// Mitsubishi GX Works2 project: 大成外環大泉FLEX   PLC: Q02/Q02H

PROGRAM FLEXPIWI  // PID演算 for WIndows
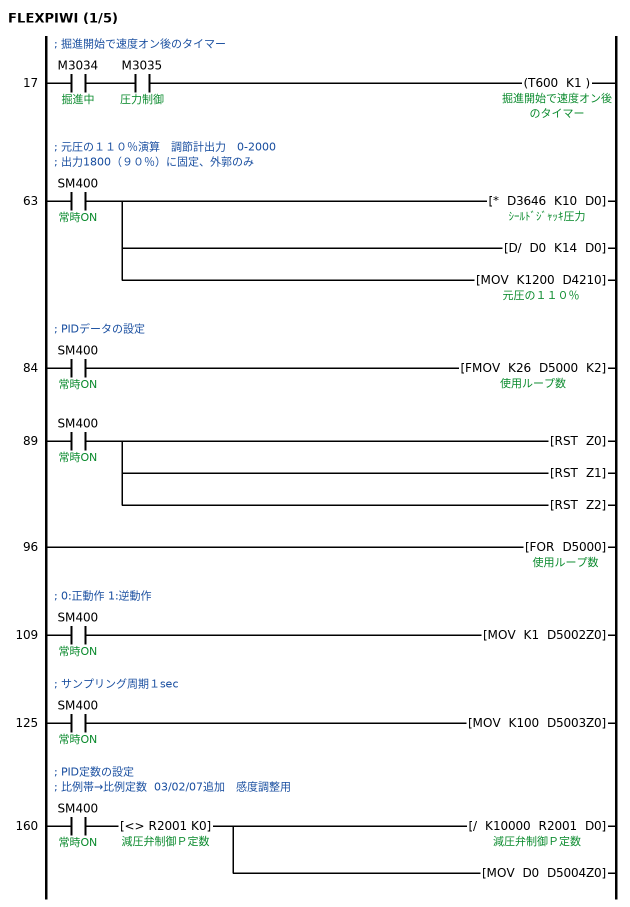
; 掘進開始で速度オン後のタイマー
17    LD      M3034  ; 掘進中
      AND     M3035  ; 圧力制御
      OUT     T600 K1  ; 掘進開始で速度オン後のタイマー
; 元圧の１１０％演算　調節計出力　0-2000
; 出力1800（９０％）に固定、外郭のみ
63    LD      SM400  ; 常時ON
      *       D3646 K10 D0  ; ｼｰﾙﾄﾞｼﾞｬｯｷ圧力
      D/      D0 K14 D0
      MOV     K1200 D4210  ; 元圧の１１０％
; PIDデータの設定
84    LD      SM400  ; 常時ON
      FMOV    K26 D5000 K2  ; 使用ループ数
89    LD      SM400  ; 常時ON
      RST     Z0
      RST     Z1
      RST     Z2
96    FOR     D5000
; 0:正動作 1:逆動作
109   LD      SM400  ; 常時ON
      MOV     K1 D5002Z0
; サンプリング周期１sec
125   LD      SM400  ; 常時ON
      MOV     K100 D5003Z0
; PID定数の設定
; 比例帯→比例定数  03/02/07追加　感度調整用
160   LD      SM400  ; 常時ON
      AND<>   R2001 K0  ; 減圧弁制御Ｐ定数
      /       K10000 R2001 D0
      MOV     D0 D5004Z0
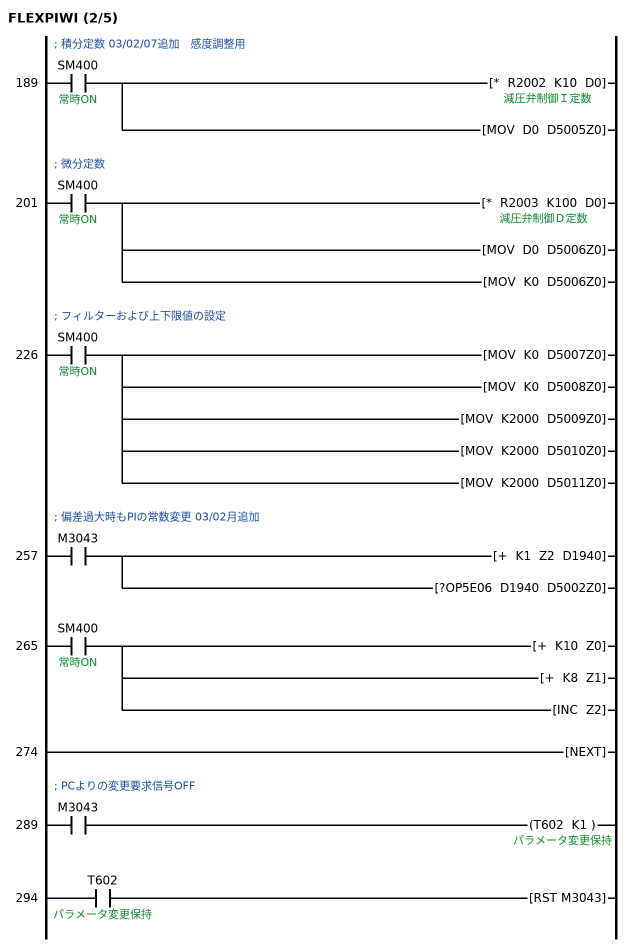
; 積分定数 03/02/07追加　感度調整用
189   LD      SM400  ; 常時ON
      *       R2002 K10 D0  ; 減圧弁制御Ｉ定数
      MOV     D0 D5005Z0
; 微分定数
201   LD      SM400  ; 常時ON
      *       R2003 K100 D0  ; 減圧弁制御Ｄ定数
      MOV     D0 D5006Z0
      MOV     K0 D5006Z0
; フィルターおよび上下限値の設定
226   LD      SM400  ; 常時ON
      MOV     K0 D5007Z0
      MOV     K0 D5008Z0
      MOV     K2000 D5009Z0
      MOV     K2000 D5010Z0
      MOV     K2000 D5011Z0
; 偏差過大時もPIの常数変更 03/02月追加
257   LD      M3043
      +       K1 Z2 D1940
      ?OP5E06 D1940 D5002Z0
265   LD      SM400  ; 常時ON
      +       K10 Z0
      +       K8 Z1
      INC     Z2
274   NEXT
; PCよりの変更要求信号OFF
289   LD      M3043
      OUT     T602 K1  ; パラメータ変更保持
294   LD      T602  ; パラメータ変更保持
      RST     M3043
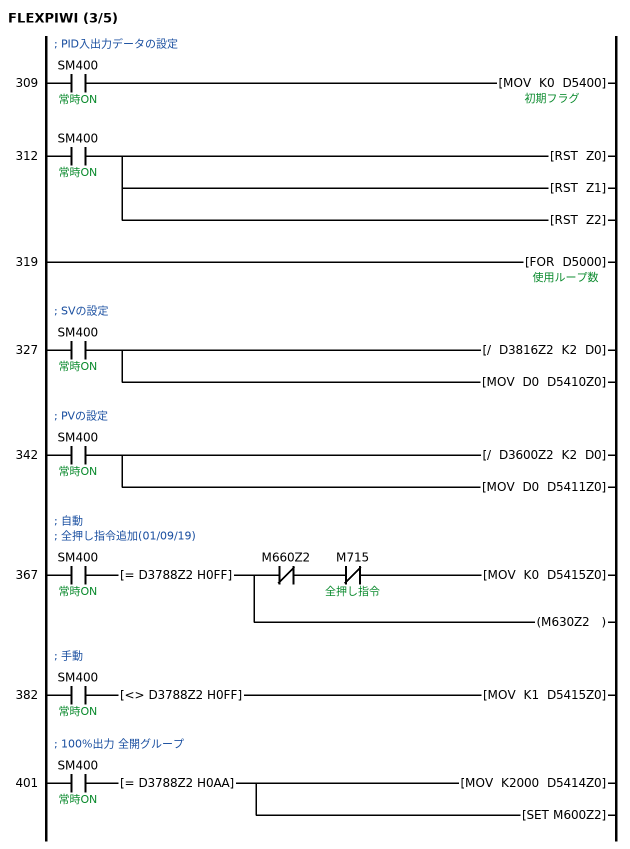
; PID入出力データの設定
309   LD      SM400  ; 常時ON
      MOV     K0 D5400  ; 初期フラグ
312   LD      SM400  ; 常時ON
      RST     Z0
      RST     Z1
      RST     Z2
319   FOR     D5000
; SVの設定
327   LD      SM400  ; 常時ON
      /       D3816Z2 K2 D0
      MOV     D0 D5410Z0
; 
; PVの設定
342   LD      SM400  ; 常時ON
      /       D3600Z2 K2 D0
      MOV     D0 D5411Z0
; 自動
; 全押し指令追加(01/09/19)
367   LD      SM400  ; 常時ON
      AND=    D3788Z2 H0FF
      MPS
      ANI     M660Z2
      ANI     M715  ; 全押し指令
      MOV     K0 D5415Z0
      MPP
      OUT     M630Z2
; 手動
382   LD      SM400  ; 常時ON
      AND<>   D3788Z2 H0FF
      MOV     K1 D5415Z0
; 100%出力 全開グループ
401   LD      SM400  ; 常時ON
      AND=    D3788Z2 H0AA
      MOV     K2000 D5414Z0
      SET     M600Z2
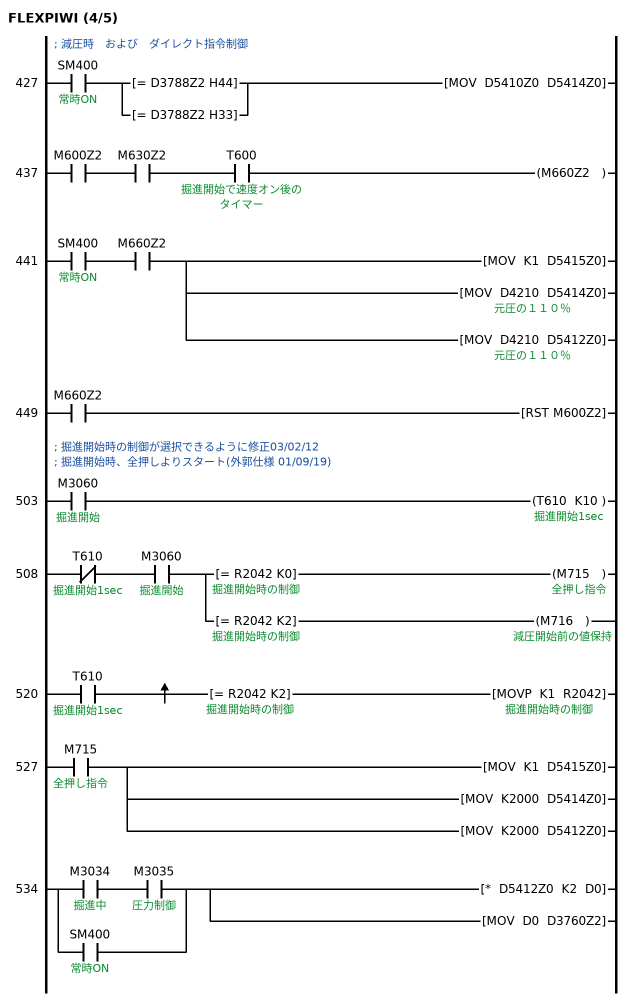
; 減圧時　および　ダイレクト指令制御
427   LD      SM400  ; 常時ON
      LD=     D3788Z2 H44
      OR=     D3788Z2 H33
      ANB
      MOV     D5410Z0 D5414Z0
437   LD      M600Z2
      AND     M630Z2
      AND     T600  ; 掘進開始で速度オン後のタイマー
      OUT     M660Z2
441   LD      SM400  ; 常時ON
      AND     M660Z2
      MOV     K1 D5415Z0
      MOV     D4210 D5414Z0
      MOV     D4210 D5412Z0
449   LD      M660Z2
      RST     M600Z2
; 掘進開始時の制御が選択できるように修正03/02/12
; 掘進開始時、全押しよりスタート(外郭仕様 01/09/19)
503   LD      M3060  ; 掘進開始
      OUT     T610 K10  ; 掘進開始1sec
508   LDI     T610  ; 掘進開始1sec
      AND     M3060  ; 掘進開始
      MPS
      AND=    R2042 K0  ; 掘進開始時の制御
      OUT     M715  ; 全押し指令
      MPP
      AND=    R2042 K2  ; 掘進開始時の制御
      OUT     M716  ; 減圧開始前の値保持
520   LD      T610  ; 掘進開始1sec
      MEP
      AND=    R2042 K2  ; 掘進開始時の制御
      MOVP    K1 R2042
527   LD      M715  ; 全押し指令
      MOV     K1 D5415Z0
      MOV     K2000 D5414Z0
      MOV     K2000 D5412Z0
534   LD      M3034  ; 掘進中
      AND     M3035  ; 圧力制御
      OR      SM400  ; 常時ON
      *       D5412Z0 K2 D0
      MOV     D0 D3760Z2
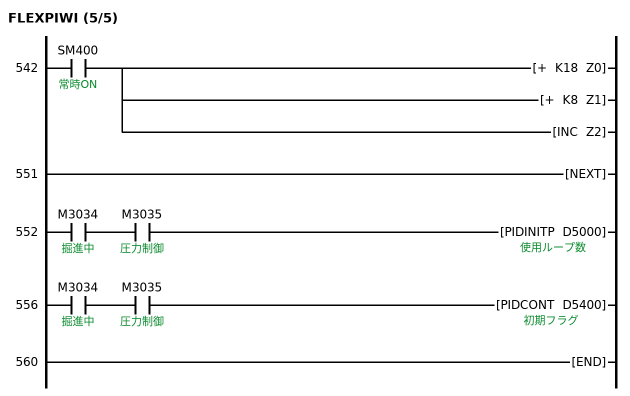
542   LD      SM400  ; 常時ON
      +       K18 Z0
      +       K8 Z1
      INC     Z2
551   NEXT
552   LD      M3034  ; 掘進中
      AND     M3035  ; 圧力制御
      PIDINITP D5000
556   LD      M3034  ; 掘進中
      AND     M3035  ; 圧力制御
      PIDCONT D5400
560   END
END_PROGRAM

PROGRAM FLEXWIN  // FlexWindos対応
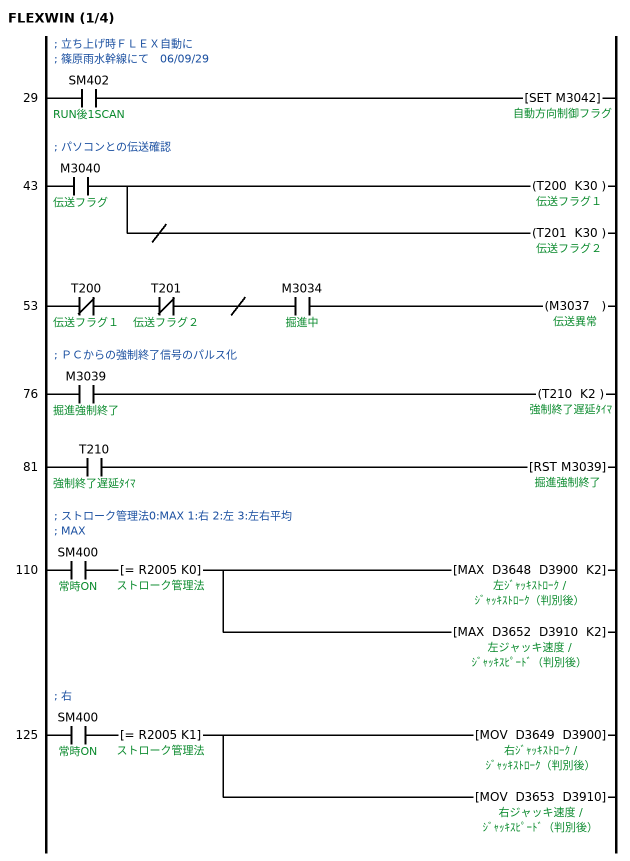
; 立ち上げ時ＦＬＥＸ自動に
; 篠原雨水幹線にて　06/09/29
29    LD      SM402  ; RUN後1SCAN
      SET     M3042  ; 自動方向制御フラグ
; パソコンとの伝送確認
43    LD      M3040  ; 伝送フラグ
      OUT     T200 K30  ; 伝送フラグ１
      INV
      OUT     T201 K30  ; 伝送フラグ２
53    LDI     T200  ; 伝送フラグ１
      ANI     T201  ; 伝送フラグ２
      INV
      AND     M3034  ; 掘進中
      OUT     M3037  ; 伝送異常
; ＰＣからの強制終了信号のパルス化
76    LD      M3039  ; 掘進強制終了
      OUT     T210 K2  ; 強制終了遅延ﾀｲﾏ
81    LD      T210  ; 強制終了遅延ﾀｲﾏ
      RST     M3039  ; 掘進強制終了
; ストローク管理法0:MAX 1:右 2:左 3:左右平均
; MAX
110   LD      SM400  ; 常時ON
      AND=    R2005 K0  ; ストローク管理法
      MAX     D3648 D3900 K2  ; 左ｼﾞｬｯｷｽﾄﾛｰｸ / ｼﾞｬｯｷｽﾄﾛｰｸ（判別後）
      MAX     D3652 D3910 K2  ; 左ジャッキ速度 / ｼﾞｬｯｷｽﾋﾟｰﾄﾞ（判別後）
; 右
125   LD      SM400  ; 常時ON
      AND=    R2005 K1  ; ストローク管理法
      MOV     D3649 D3900  ; 右ｼﾞｬｯｷｽﾄﾛｰｸ
      MOV     D3653 D3910  ; 右ジャッキ速度
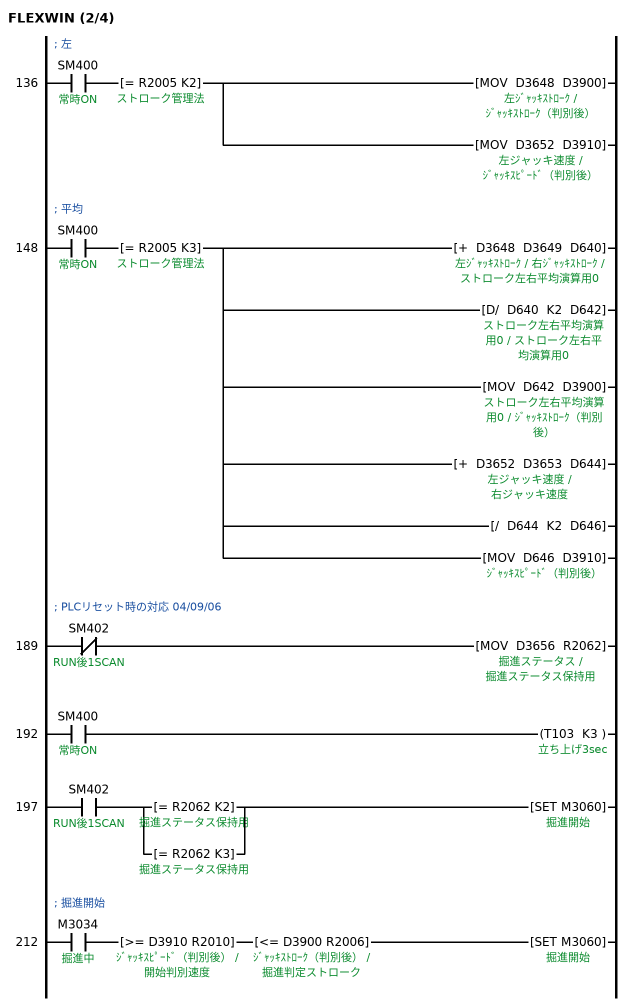
; 左
136   LD      SM400  ; 常時ON
      AND=    R2005 K2  ; ストローク管理法
      MOV     D3648 D3900
      MOV     D3652 D3910
; 平均
148   LD      SM400  ; 常時ON
      AND=    R2005 K3  ; ストローク管理法
      +       D3648 D3649 D640  ; ストローク左右平均演算用0
      D/      D640 K2 D642  ; ストローク左右平均演算用0
      MOV     D642 D3900
      +       D3652 D3653 D644
      /       D644 K2 D646
      MOV     D646 D3910
; PLCリセット時の対応 04/09/06
189   LDI     SM402  ; RUN後1SCAN
      MOV     D3656 R2062  ; 掘進ステータス / 掘進ステータス保持用
192   LD      SM400  ; 常時ON
      OUT     T103 K3  ; 立ち上げ3sec
197   LD      SM402  ; RUN後1SCAN
      LD=     R2062 K2  ; 掘進ステータス保持用
      OR=     R2062 K3  ; 掘進ステータス保持用
      ANB
      SET     M3060  ; 掘進開始
; 掘進開始
212   LD      M3034  ; 掘進中
      AND>=   D3910 R2010  ; ｼﾞｬｯｷｽﾋﾟｰﾄﾞ（判別後） / 開始判別速度
      AND<=   D3900 R2006  ; ｼﾞｬｯｷｽﾄﾛｰｸ（判別後） / 掘進判定ストローク
      SET     M3060  ; 掘進開始
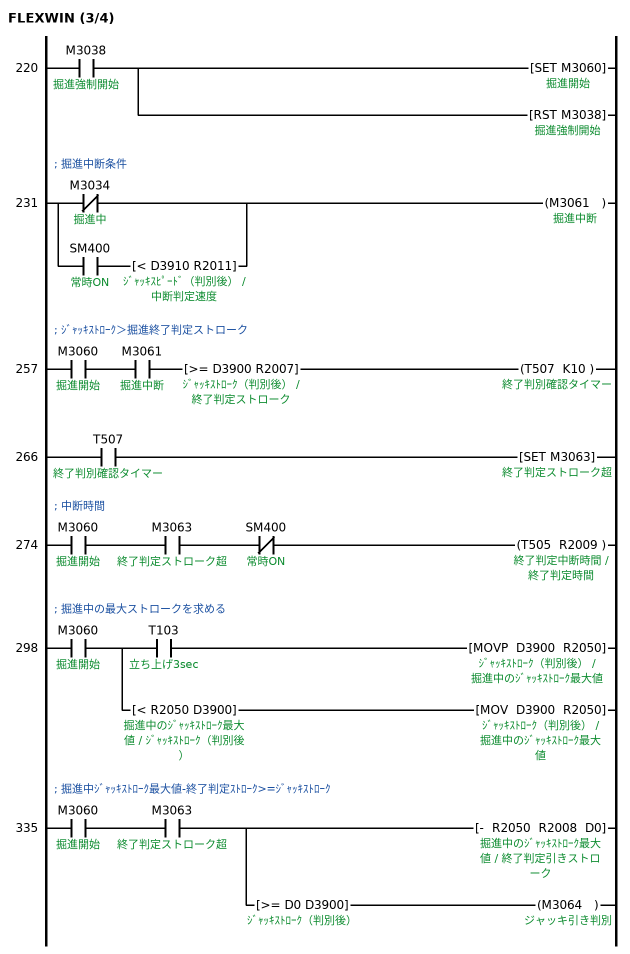
220   LD      M3038  ; 掘進強制開始
      SET     M3060  ; 掘進開始
      RST     M3038  ; 掘進強制開始
; 掘進中断条件
231   LDI     M3034  ; 掘進中
      LD      SM400  ; 常時ON
      AND<    D3910 R2011  ; ｼﾞｬｯｷｽﾋﾟｰﾄﾞ（判別後） / 中断判定速度
      ORB
      OUT     M3061  ; 掘進中断
; ｼﾞｬｯｷｽﾄﾛｰｸ＞掘進終了判定ストローク
257   LD      M3060  ; 掘進開始
      AND     M3061  ; 掘進中断
      AND>=   D3900 R2007  ; ｼﾞｬｯｷｽﾄﾛｰｸ（判別後） / 終了判定ストローク
      OUT     T507 K10  ; 終了判別確認タイマー
266   LD      T507  ; 終了判別確認タイマー
      SET     M3063  ; 終了判定ストローク超
; 中断時間
274   LD      M3060  ; 掘進開始
      AND     M3063  ; 終了判定ストローク超
      ANI     SM400  ; 常時ON
      OUT     T505 R2009  ; 終了判定中断時間 / 終了判定時間
; 掘進中の最大ストロークを求める
298   LD      M3060  ; 掘進開始
      MPS
      AND     T103  ; 立ち上げ3sec
      MOVP    D3900 R2050  ; 掘進中のｼﾞｬｯｷｽﾄﾛｰｸ最大値
      MPP
      AND<    R2050 D3900  ; 掘進中のｼﾞｬｯｷｽﾄﾛｰｸ最大値 / ｼﾞｬｯｷｽﾄﾛｰｸ（判別後）
      MOV     D3900 R2050
; 掘進中ｼﾞｬｯｷｽﾄﾛｰｸ最大値-終了判定ｽﾄﾛｰｸ>=ｼﾞｬｯｷｽﾄﾛｰｸ
335   LD      M3060  ; 掘進開始
      AND     M3063  ; 終了判定ストローク超
      -       R2050 R2008 D0  ; 終了判定引きストローク
      AND>=   D0 D3900  ; ｼﾞｬｯｷｽﾄﾛｰｸ（判別後）
      OUT     M3064  ; ジャッキ引き判別
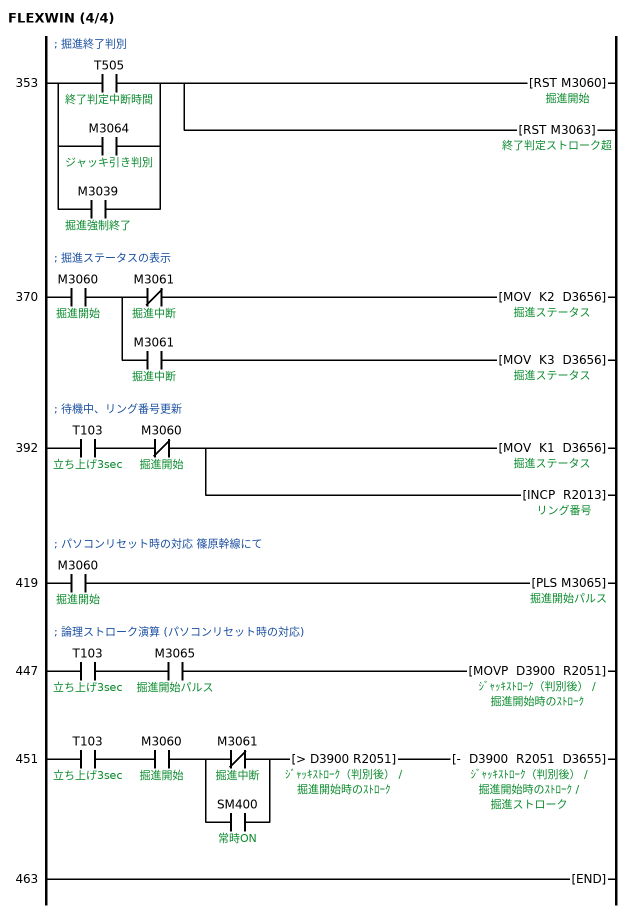
; 掘進終了判別
353   LD      T505  ; 終了判定中断時間
      OR      M3064  ; ジャッキ引き判別
      OR      M3039  ; 掘進強制終了
      RST     M3060  ; 掘進開始
      RST     M3063  ; 終了判定ストローク超
; 掘進ステータスの表示
370   LD      M3060  ; 掘進開始
      MPS
      ANI     M3061  ; 掘進中断
      MOV     K2 D3656
      MPP
      AND     M3061  ; 掘進中断
      MOV     K3 D3656
; 待機中、リング番号更新
392   LD      T103  ; 立ち上げ3sec
      ANI     M3060  ; 掘進開始
      MOV     K1 D3656
      INCP    R2013  ; リング番号
; パソコンリセット時の対応 篠原幹線にて
419   LD      M3060  ; 掘進開始
      PLS     M3065  ; 掘進開始パルス
; 論理ストローク演算 (パソコンリセット時の対応)
447   LD      T103  ; 立ち上げ3sec
      AND     M3065  ; 掘進開始パルス
      MOVP    D3900 R2051  ; 掘進開始時のｽﾄﾛｰｸ
451   LD      T103  ; 立ち上げ3sec
      AND     M3060  ; 掘進開始
      LDI     M3061  ; 掘進中断
      OR      SM400  ; 常時ON
      ANB
      AND>    D3900 R2051  ; ｼﾞｬｯｷｽﾄﾛｰｸ（判別後） / 掘進開始時のｽﾄﾛｰｸ
      -       D3900 R2051 D3655  ; 掘進ストローク
463   END
END_PROGRAM

PROGRAM INOUTWIN  // 大成外環大泉FLEX
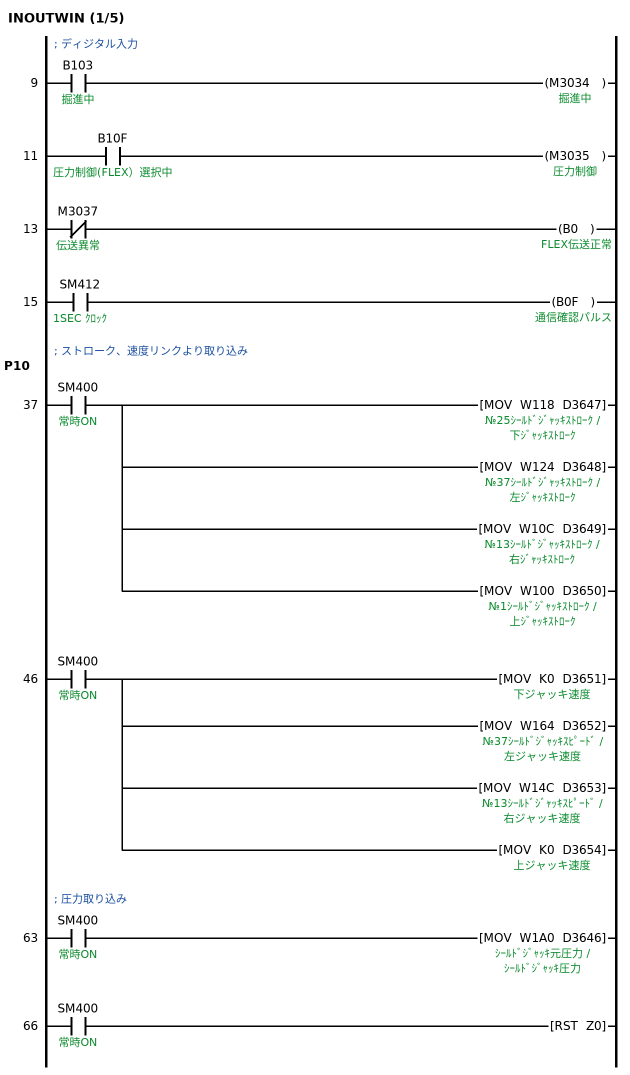
; ディジタル入力
9     LD      B103  ; 掘進中
      OUT     M3034  ; 掘進中
11    LD      B10F  ; 圧力制御(FLEX）選択中
      OUT     M3035  ; 圧力制御
13    LDI     M3037  ; 伝送異常
      OUT     B0  ; FLEX伝送正常
15    LD      SM412  ; 1SEC ｸﾛｯｸ
      OUT     B0F  ; 通信確認パルス
; ストローク、速度リンクより取り込み
      P10
37    LD      SM400  ; 常時ON
      MOV     W118 D3647  ; №25ｼｰﾙﾄﾞｼﾞｬｯｷｽﾄﾛｰｸ / 下ｼﾞｬｯｷｽﾄﾛｰｸ
      MOV     W124 D3648  ; №37ｼｰﾙﾄﾞｼﾞｬｯｷｽﾄﾛｰｸ / 左ｼﾞｬｯｷｽﾄﾛｰｸ
      MOV     W10C D3649  ; №13ｼｰﾙﾄﾞｼﾞｬｯｷｽﾄﾛｰｸ / 右ｼﾞｬｯｷｽﾄﾛｰｸ
      MOV     W100 D3650  ; №1ｼｰﾙﾄﾞｼﾞｬｯｷｽﾄﾛｰｸ / 上ｼﾞｬｯｷｽﾄﾛｰｸ
46    LD      SM400  ; 常時ON
      MOV     K0 D3651  ; 下ジャッキ速度
      MOV     W164 D3652  ; №37ｼｰﾙﾄﾞｼﾞｬｯｷｽﾋﾟｰﾄﾞ / 左ジャッキ速度
      MOV     W14C D3653  ; №13ｼｰﾙﾄﾞｼﾞｬｯｷｽﾋﾟｰﾄﾞ / 右ジャッキ速度
      MOV     K0 D3654  ; 上ジャッキ速度
; 圧力取り込み
63    LD      SM400  ; 常時ON
      MOV     W1A0 D3646  ; ｼｰﾙﾄﾞｼﾞｬｯｷ元圧力 / ｼｰﾙﾄﾞｼﾞｬｯｷ圧力
66    LD      SM400  ; 常時ON
      RST     Z0
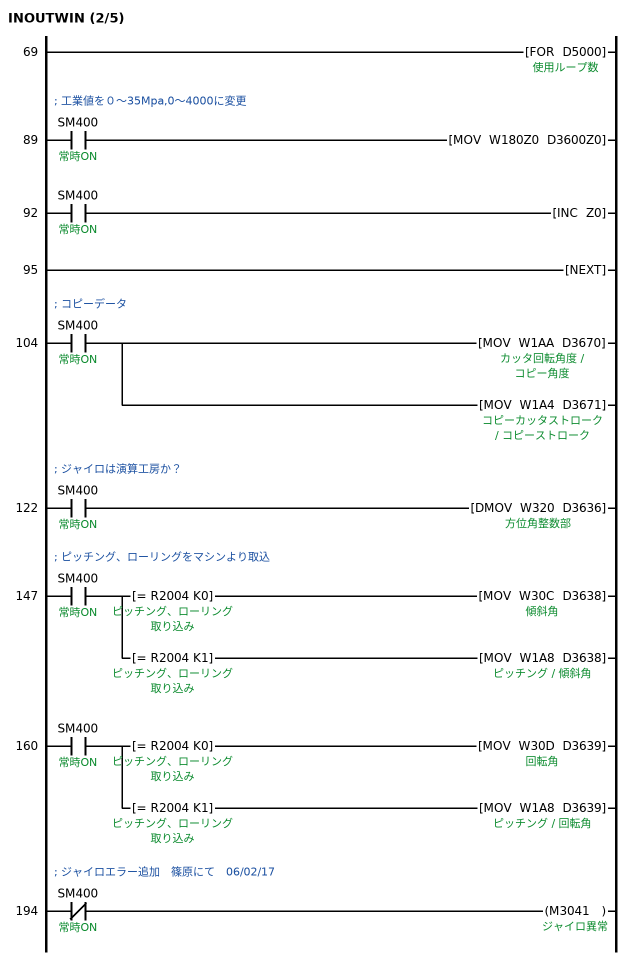
69    FOR     D5000  ; 使用ループ数
; 工業値を０～35Mpa,0～4000に変更
89    LD      SM400  ; 常時ON
      MOV     W180Z0 D3600Z0
92    LD      SM400  ; 常時ON
      INC     Z0
95    NEXT
; コピーデータ
104   LD      SM400  ; 常時ON
      MOV     W1AA D3670  ; カッタ回転角度 / コピー角度
      MOV     W1A4 D3671  ; コピーカッタストローク / コピーストローク
; ジャイロは演算工房か？
122   LD      SM400  ; 常時ON
      DMOV    W320 D3636  ; 方位角整数部
; ピッチング、ローリングをマシンより取込
147   LD      SM400  ; 常時ON
      MPS
      AND=    R2004 K0  ; ピッチング、ローリング取り込み
      MOV     W30C D3638  ; 傾斜角
      MPP
      AND=    R2004 K1  ; ピッチング、ローリング取り込み
      MOV     W1A8 D3638  ; ピッチング
160   LD      SM400  ; 常時ON
      MPS
      AND=    R2004 K0  ; ピッチング、ローリング取り込み
      MOV     W30D D3639  ; 回転角
      MPP
      AND=    R2004 K1  ; ピッチング、ローリング取り込み
      MOV     W1A8 D3639
; ジャイロエラー追加　篠原にて　06/02/17
194   LDI     SM400  ; 常時ON
      OUT     M3041  ; ジャイロ異常
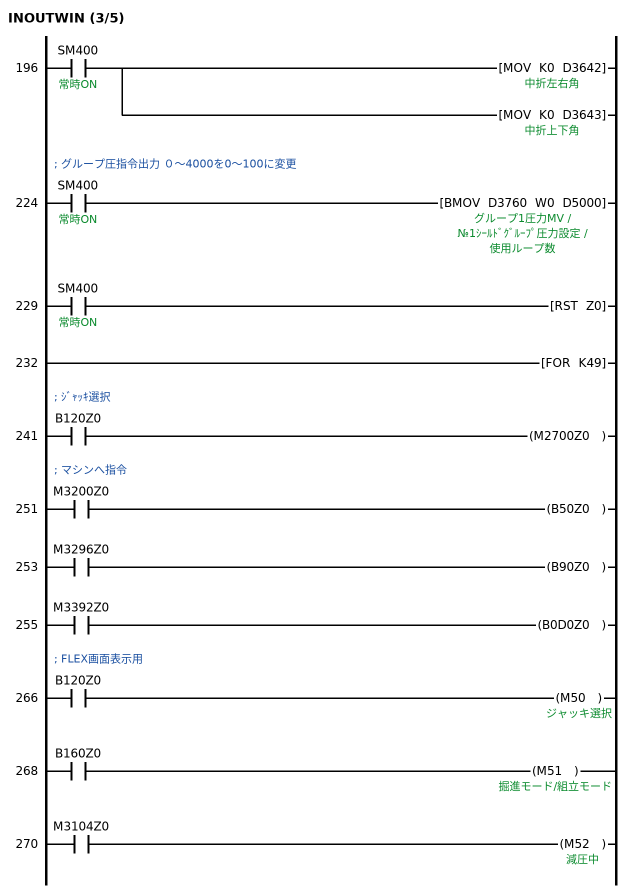
196   LD      SM400  ; 常時ON
      MOV     K0 D3642  ; 中折左右角
      MOV     K0 D3643  ; 中折上下角
; グループ圧指令出力 ０～4000を0～100に変更
224   LD      SM400  ; 常時ON
      BMOV    D3760 W0 D5000  ; グループ1圧力MV / №1ｼｰﾙﾄﾞｸﾞﾙｰﾌﾟ圧力設定
229   LD      SM400  ; 常時ON
      RST     Z0
232   FOR     K49
; ｼﾞｬｯｷ選択
241   LD      B120Z0
      OUT     M2700Z0
; マシンへ指令
251   LD      M3200Z0
      OUT     B50Z0
253   LD      M3296Z0
      OUT     B90Z0
255   LD      M3392Z0
      OUT     B0D0Z0
; FLEX画面表示用
266   LD      B120Z0
      OUT     M50  ; ジャッキ選択
268   LD      B160Z0
      OUT     M51  ; 掘進モード/組立モード
270   LD      M3104Z0
      OUT     M52  ; 減圧中
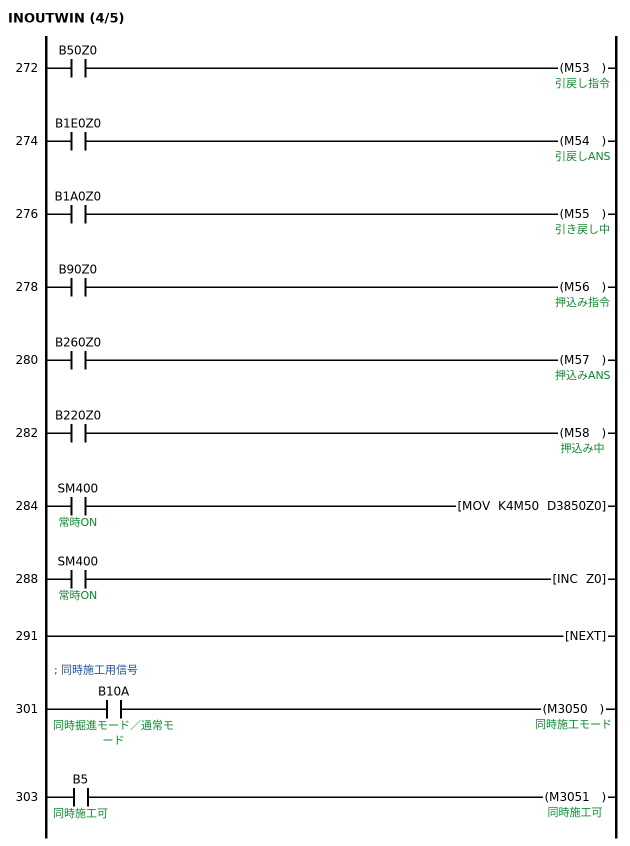
272   LD      B50Z0
      OUT     M53  ; 引戻し指令
274   LD      B1E0Z0
      OUT     M54  ; 引戻しANS
276   LD      B1A0Z0
      OUT     M55  ; 引き戻し中
278   LD      B90Z0
      OUT     M56  ; 押込み指令
280   LD      B260Z0
      OUT     M57  ; 押込みANS
282   LD      B220Z0
      OUT     M58  ; 押込み中
284   LD      SM400  ; 常時ON
      MOV     K4M50 D3850Z0
288   LD      SM400  ; 常時ON
      INC     Z0
291   NEXT
; 同時施工用信号
301   LD      B10A  ; 同時掘進モード／通常モード
      OUT     M3050  ; 同時施工モード
303   LD      B5  ; 同時施工可
      OUT     M3051  ; 同時施工可
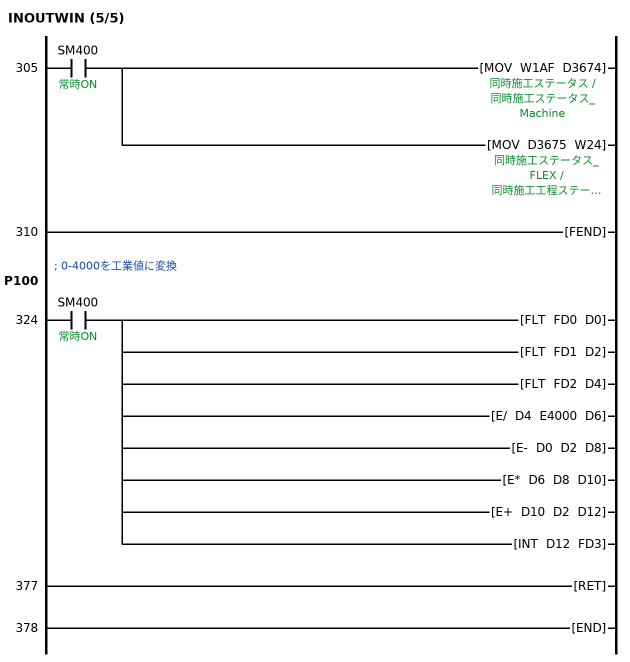
305   LD      SM400  ; 常時ON
      MOV     W1AF D3674  ; 同時施工ステータス / 同時施工ステータス_Machine
      MOV     D3675 W24  ; 同時施工ステータス_FLEX / 同時施工工程ステータス
310   FEND
      P100
; 0-4000を工業値に変換
324   LD      SM400  ; 常時ON
      FLT     FD0 D0
        [note] スケール上限
      FLT     FD1 D2
        [note] スケール下限
      FLT     FD2 D4
        [note] 元アドレス
      E/      D4 E4000 D6
      E-      D0 D2 D8
      E*      D6 D8 D10
      E+      D10 D2 D12
      INT     D12 FD3
377   RET
378   END
END_PROGRAM

PROGRAM TOKIMEC  // ジャイロとの通信 QJ71C24Nタ
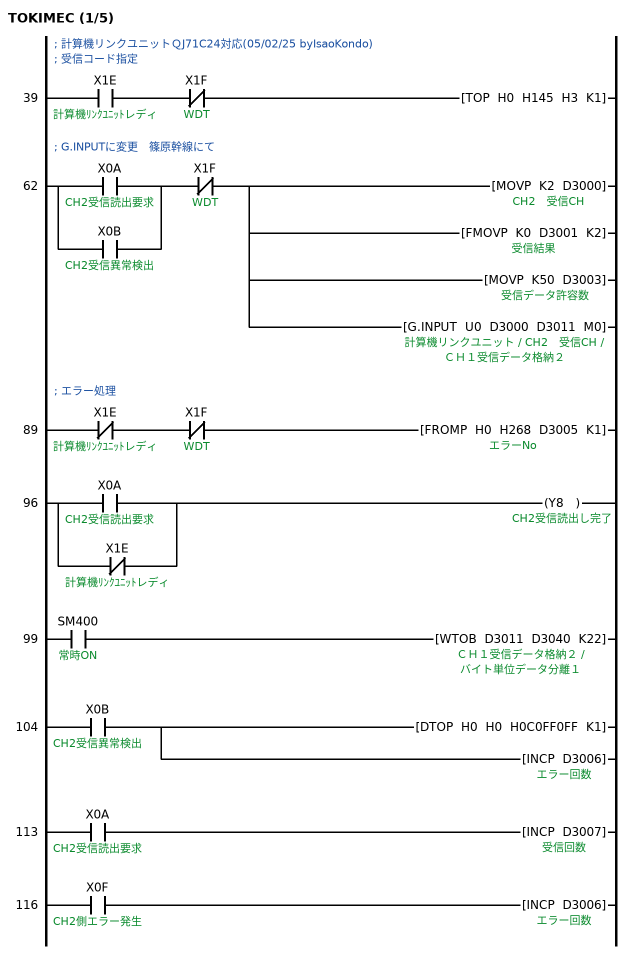
; 計算機リンクユニットＱJ71C24対応(05/02/25 byIsaoKondo)
; 受信コード指定
39    LD      X1E  ; 計算機ﾘﾝｸﾕﾆｯﾄレディ
      ANI     X1F  ; WDT
      TOP     H0 H145 H3 K1
; G.INPUTに変更　篠原幹線にて
62    LD      X0A  ; CH2受信読出要求
      OR      X0B  ; CH2受信異常検出
      ANI     X1F  ; WDT
      MOVP    K2 D3000  ; CH2　受信CH
      FMOVP   K0 D3001 K2  ; 受信結果
      MOVP    K50 D3003  ; 受信データ許容数
      G.INPUT U0 D3000 D3011 M0  ; 計算機リンクユニット / ＣＨ１受信データ格納２
; エラー処理
89    LDI     X1E  ; 計算機ﾘﾝｸﾕﾆｯﾄレディ
      ANI     X1F  ; WDT
      FROMP   H0 H268 D3005 K1  ; エラーNo
96    LD      X0A  ; CH2受信読出要求
      ORI     X1E  ; 計算機ﾘﾝｸﾕﾆｯﾄレディ
      OUT     Y8  ; CH2受信読出し完了
99    LD      SM400  ; 常時ON
      WTOB    D3011 D3040 K22  ; バイト単位データ分離１
104   LD      X0B  ; CH2受信異常検出
      DTOP    H0 H0 H0C0FF0FF K1
      INCP    D3006  ; エラー回数
113   LD      X0A  ; CH2受信読出要求
      INCP    D3007  ; 受信回数
116   LD      X0F  ; CH2側エラー発生
      INCP    D3006
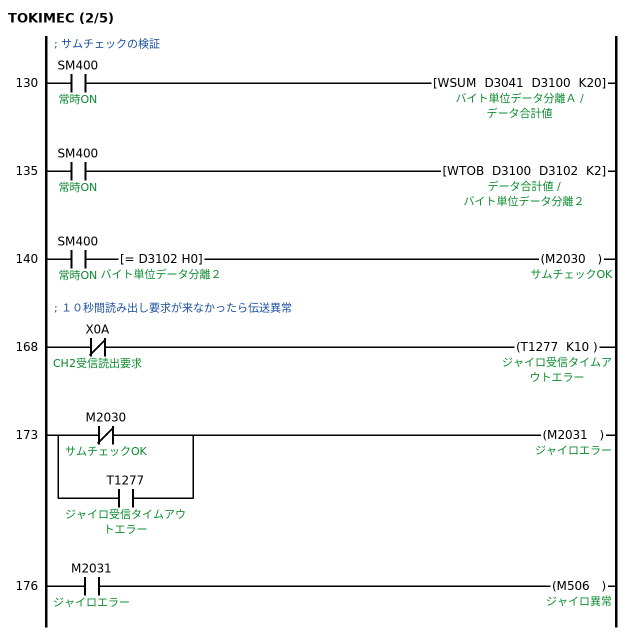
; サムチェックの検証
130   LD      SM400  ; 常時ON
      WSUM    D3041 D3100 K20  ; バイト単位データ分離Ａ / データ合計値
135   LD      SM400  ; 常時ON
      WTOB    D3100 D3102 K2  ; バイト単位データ分離２
140   LD      SM400  ; 常時ON
      AND=    D3102 H0  ; バイト単位データ分離２
      OUT     M2030  ; サムチェックOK
; １０秒間読み出し要求が来なかったら伝送異常
168   LDI     X0A  ; CH2受信読出要求
      OUT     T1277 K10  ; ジャイロ受信タイムアウトエラー
173   LDI     M2030  ; サムチェックOK
      OR      T1277  ; ジャイロ受信タイムアウトエラー
      OUT     M2031  ; ジャイロエラー
176   LD      M2031  ; ジャイロエラー
      OUT     M506  ; ジャイロ異常
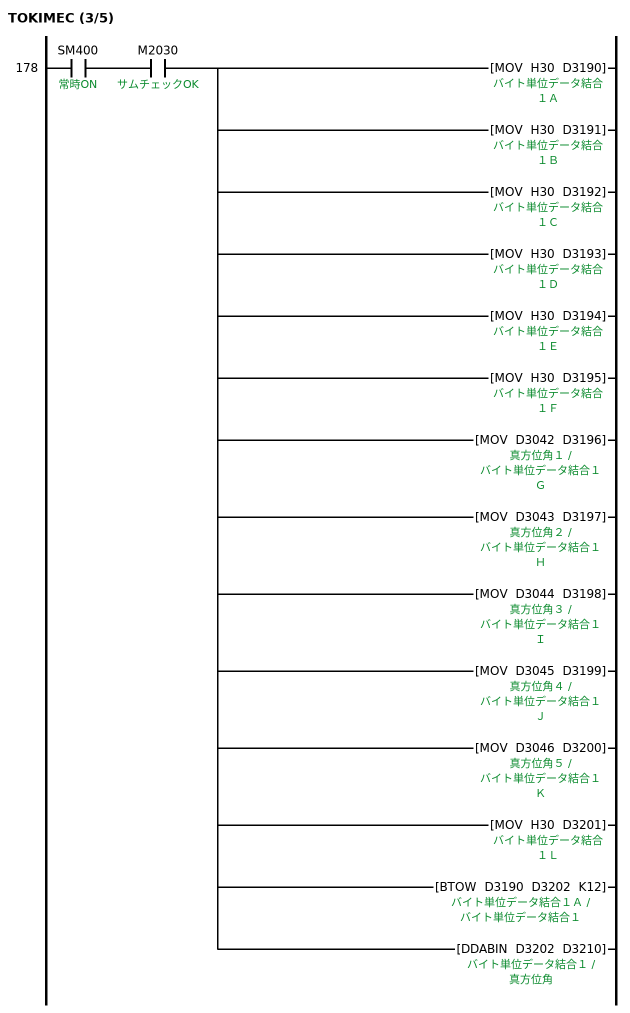
178   LD      SM400  ; 常時ON
      AND     M2030  ; サムチェックOK
      MOV     H30 D3190  ; バイト単位データ結合１Ａ
      MOV     H30 D3191  ; バイト単位データ結合１Ｂ
      MOV     H30 D3192  ; バイト単位データ結合１Ｃ
      MOV     H30 D3193  ; バイト単位データ結合１Ｄ
      MOV     H30 D3194  ; バイト単位データ結合１Ｅ
      MOV     H30 D3195  ; バイト単位データ結合１Ｆ
      MOV     D3042 D3196  ; 真方位角１ / バイト単位データ結合１Ｇ
      MOV     D3043 D3197  ; 真方位角２ / バイト単位データ結合１Ｈ
      MOV     D3044 D3198  ; 真方位角３ / バイト単位データ結合１Ｉ
      MOV     D3045 D3199  ; 真方位角４ / バイト単位データ結合１Ｊ
      MOV     D3046 D3200  ; 真方位角５ / バイト単位データ結合１Ｋ
      MOV     H30 D3201  ; バイト単位データ結合１Ｌ
      BTOW    D3190 D3202 K12  ; バイト単位データ結合１
      DDABIN  D3202 D3210  ; 真方位角
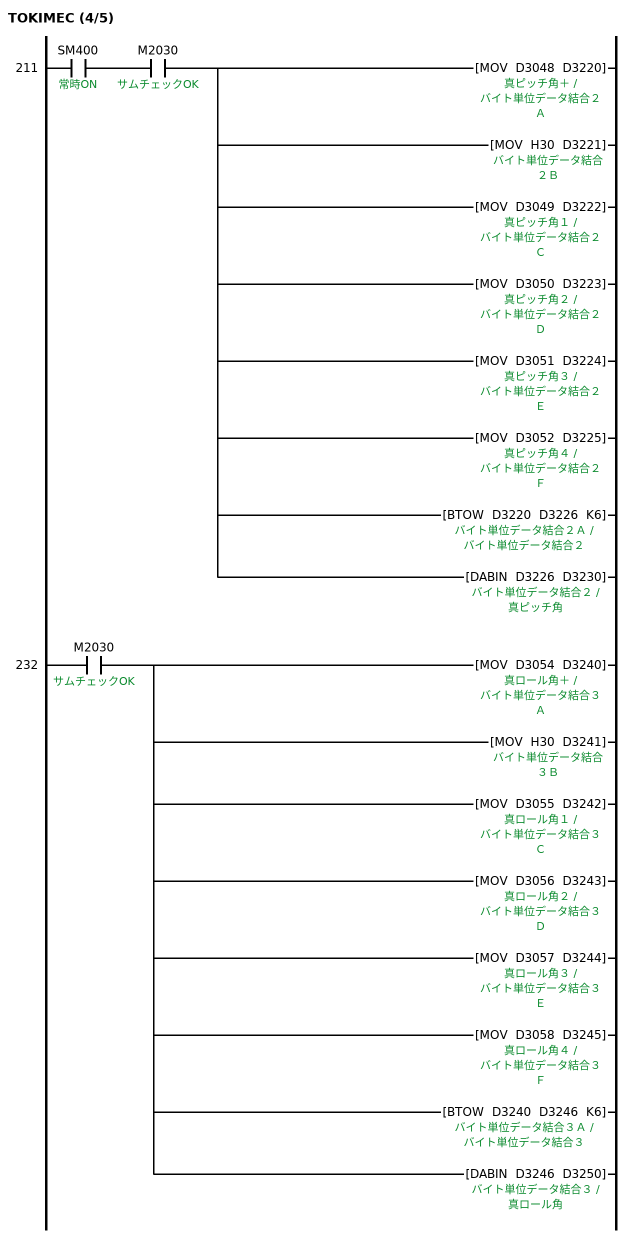
211   LD      SM400  ; 常時ON
      AND     M2030  ; サムチェックOK
      MOV     D3048 D3220  ; 真ピッチ角＋ / バイト単位データ結合２Ａ
      MOV     H30 D3221  ; バイト単位データ結合２Ｂ
      MOV     D3049 D3222  ; 真ピッチ角１ / バイト単位データ結合２Ｃ
      MOV     D3050 D3223  ; 真ピッチ角２ / バイト単位データ結合２Ｄ
      MOV     D3051 D3224  ; 真ピッチ角３ / バイト単位データ結合２Ｅ
      MOV     D3052 D3225  ; 真ピッチ角４ / バイト単位データ結合２Ｆ
      BTOW    D3220 D3226 K6  ; バイト単位データ結合２
      DABIN   D3226 D3230  ; 真ピッチ角
232   LD      M2030  ; サムチェックOK
      MOV     D3054 D3240  ; 真ロール角＋ / バイト単位データ結合３Ａ
      MOV     H30 D3241  ; バイト単位データ結合３Ｂ
      MOV     D3055 D3242  ; 真ロール角１ / バイト単位データ結合３Ｃ
      MOV     D3056 D3243  ; 真ロール角２ / バイト単位データ結合３Ｄ
      MOV     D3057 D3244  ; 真ロール角３ / バイト単位データ結合３Ｅ
      MOV     D3058 D3245  ; 真ロール角４ / バイト単位データ結合３Ｆ
      BTOW    D3240 D3246 K6  ; バイト単位データ結合３
      DABIN   D3246 D3250  ; 真ロール角
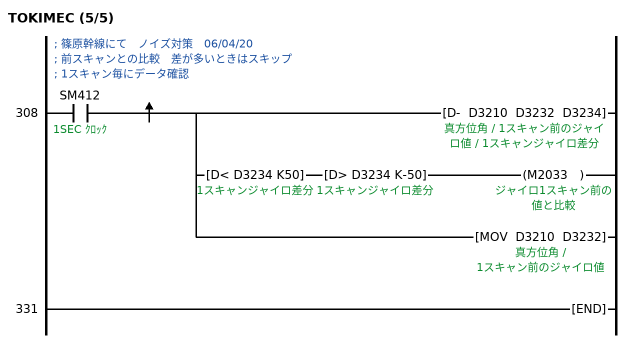
; 篠原幹線にて　ノイズ対策　06/04/20
; 前スキャンとの比較　差が多いときはスキップ
; 1スキャン毎にデータ確認
308   LD      SM412  ; 1SEC ｸﾛｯｸ
      MEP
      D-      D3210 D3232 D3234  ; 1スキャン前のジャイロ値 / 1スキャンジャイロ差分
      MPS
      ANDD<   D3234 K50  ; 1スキャンジャイロ差分
      ANDD>   D3234 K-50  ; 1スキャンジャイロ差分
      OUT     M2033  ; ジャイロ1スキャン前の値と比較
      MPP
      MOV     D3210 D3232
331   END
END_PROGRAM

PROGRAM Simlat  // 大成外環シュミレーション
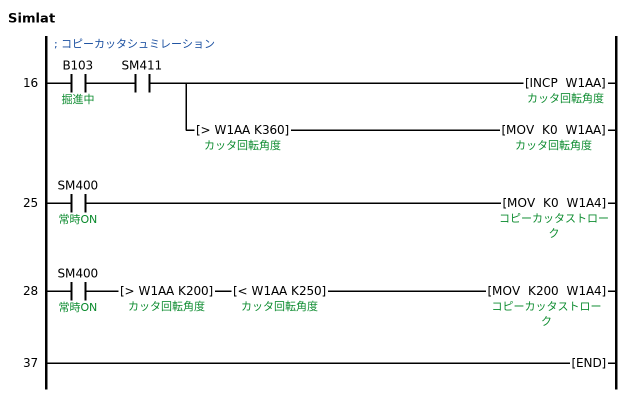
; コピーカッタシュミレーション
16    LD      B103  ; 掘進中
      AND     SM411
      INCP    W1AA  ; カッタ回転角度
      AND>    W1AA K360  ; カッタ回転角度
      MOV     K0 W1AA
25    LD      SM400  ; 常時ON
      MOV     K0 W1A4  ; コピーカッタストローク
28    LD      SM400  ; 常時ON
      AND>    W1AA K200  ; カッタ回転角度
      AND<    W1AA K250  ; カッタ回転角度
      MOV     K200 W1A4
37    END
END_PROGRAM

// device comments not shown above
D3600  ; グループ1圧力
D3816  ; グループ1圧力SV
D5002  ; グループ1演算式選択
D5412  ; グループ1自動操作量（MV)
